// TIA Portal V19 export
TYPE "LAF_typeInterfaceSignals"
TITLE = Structure of interface signals / Struktur Schnittstellen Signale
// This type is for combining the symbolic name with the status of the variable for the boolean interface functionality. / Interface signals
// stored: Access Published
   STRUCT
      value : Bool;   // HMI: Aktueller Zustand des Signals / HMI: Current state of signals
      symbolName : WString[60];   // HMI: Symbolischer Name des Signals / HMI: Symbolic name of signal
   END_STRUCT;
END_TYPE
